// TIA Portal V17 export
// export: Created 2024-09-02T12:50:23.7174179Z, ExportSetting WithDefaults, DisplayName Totally Integrated Automation Portal, DisplayVersion V17, DisplayName TIA Portal Openness, DisplayVersion V17, DisplayName TIA Portal Version Control Interface, DisplayVersion V17, DisplayName STEP 7 Professional, DisplayVersion V17, DisplayName STEP 7 Safety, DisplayVersion V17, DisplayName WinCC Professional, DisplayVersion V17
FUNCTION "AnwFC_StatusStation_OP70" : Void   // FC43, LAD
{ S7_Optimized_Access := 'TRUE' }
VERSION : 0.1
// stored: AutoNumber true, IsIECCheckEnabled false, SetENOAutomatically false, UDAEnableTagReadback false
   VAR_TEMP   // added for the SCL form of the ladder/FBD networks
      _w1 : Bool;
   END_VAR
BEGIN

REGION Network 1: Station Status signals
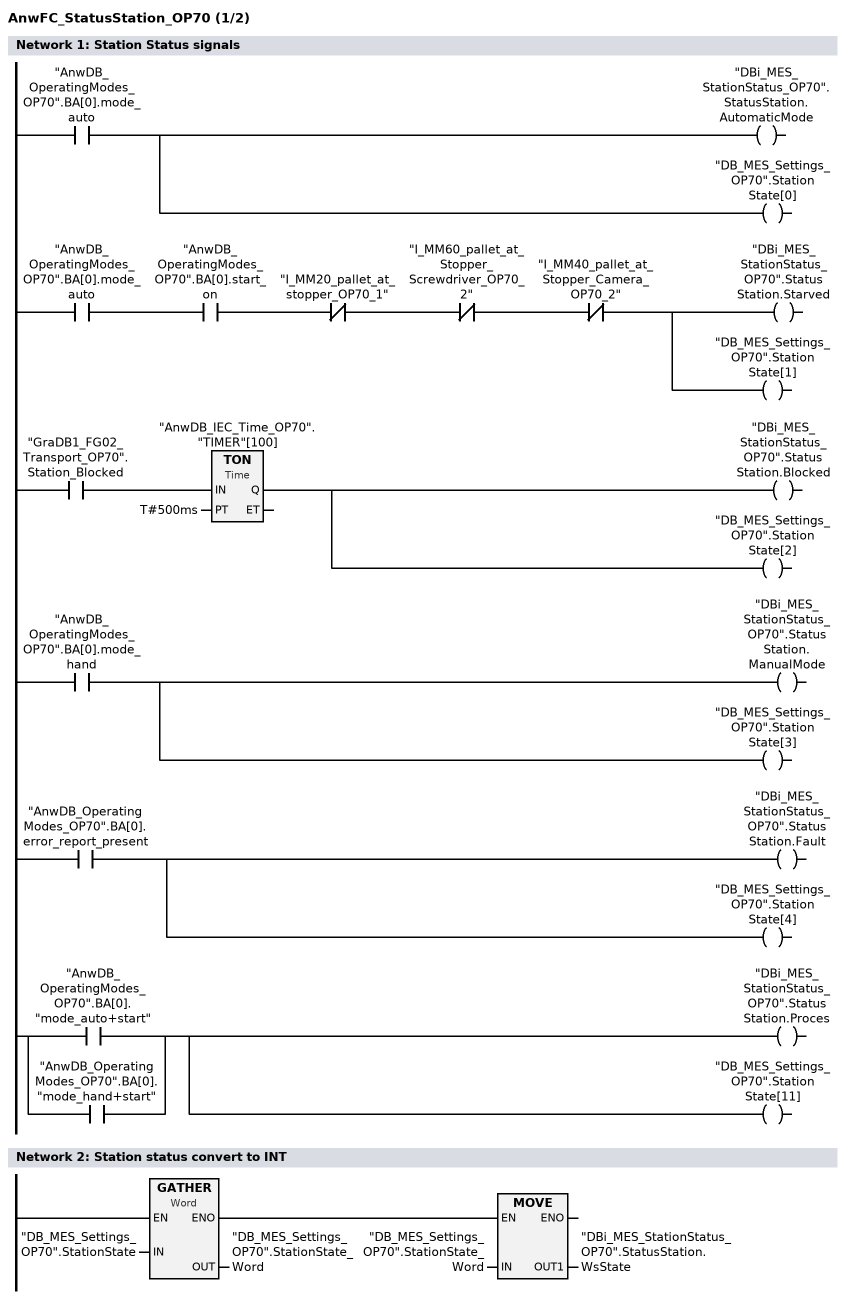
   RUNG wire#powerrail
      Contact( "AnwDB_OperatingModes_OP70".BA[0].mode_auto )
      wire#w1
      Coil( "DBi_MES_StationStatus_OP70".StatusStation.AutomaticMode )
   END_RUNG
   RUNG wire#w1
      Coil( "DB_MES_Settings_OP70".StationState[0] )
   END_RUNG
   RUNG wire#powerrail
      Contact( "AnwDB_OperatingModes_OP70".BA[0].mode_auto )
      Contact( "AnwDB_OperatingModes_OP70".BA[0].start_on )
      I_Contact( "I_MM20_pallet_at_stopper_OP70_1" )
      I_Contact( "I_MM60_pallet_at_Stopper_Screwdriver_OP70_2" )
      I_Contact( "I_MM40_pallet_at_Stopper_Camera_OP70_2" )
      wire#w2
      Coil( "DBi_MES_StationStatus_OP70".StatusStation.Starved )
   END_RUNG
   RUNG wire#w2
      Coil( "DB_MES_Settings_OP70".StationState[1] )
   END_RUNG
   RUNG wire#powerrail
      Contact( "GraDB1_FG02_Transport_OP70".Station_Blocked )
      { S7_Templates := "time_type := Time" } "AnwDB_IEC_Time_OP70"."TIMER"[100].TON(pt := T#500ms, et =>)
      wire#w3
      Coil( "DBi_MES_StationStatus_OP70".StatusStation.Blocked )
   END_RUNG
   RUNG wire#w3
      Coil( "DB_MES_Settings_OP70".StationState[2] )
   END_RUNG
   RUNG wire#powerrail
      Contact( "AnwDB_OperatingModes_OP70".BA[0].mode_hand )
      wire#w4
      Coil( "DBi_MES_StationStatus_OP70".StatusStation.ManualMode )
   END_RUNG
   RUNG wire#w4
      Coil( "DB_MES_Settings_OP70".StationState[3] )
   END_RUNG
   RUNG wire#powerrail
      Contact( "AnwDB_OperatingModes_OP70".BA[0].error_report_present )
      wire#w5
      Coil( "DBi_MES_StationStatus_OP70".StatusStation.Fault )
   END_RUNG
   RUNG wire#w5
      Coil( "DB_MES_Settings_OP70".StationState[4] )
   END_RUNG
   RUNG wire#powerrail
      Contact( "AnwDB_OperatingModes_OP70".BA[0]."mode_auto+start" )
      wire#w6
      Coil( "DBi_MES_StationStatus_OP70".StatusStation.Proces )
   END_RUNG
   RUNG wire#powerrail
      Contact( "AnwDB_OperatingModes_OP70".BA[0]."mode_hand+start" )
   END_RUNG wire#w6
   RUNG wire#w6
      Coil( "DB_MES_Settings_OP70".StationState[11] )
   END_RUNG
   // the same network as SCL:
   "DBi_MES_StationStatus_OP70".StatusStation.AutomaticMode := "AnwDB_OperatingModes_OP70".BA[0].mode_auto;
   "DB_MES_Settings_OP70".StationState[0] := "AnwDB_OperatingModes_OP70".BA[0].mode_auto;
   "DBi_MES_StationStatus_OP70".StatusStation.Starved := "AnwDB_OperatingModes_OP70".BA[0].mode_auto AND "AnwDB_OperatingModes_OP70".BA[0].start_on AND NOT "I_MM20_pallet_at_stopper_OP70_1" AND NOT "I_MM60_pallet_at_Stopper_Screwdriver_OP70_2" AND NOT "I_MM40_pallet_at_Stopper_Camera_OP70_2";
   "DB_MES_Settings_OP70".StationState[1] := "DBi_MES_StationStatus_OP70".StatusStation.Starved;
   "AnwDB_IEC_Time_OP70"."TIMER"[100].TON(IN := "GraDB1_FG02_Transport_OP70".Station_Blocked, PT := T#500ms);
   "DBi_MES_StationStatus_OP70".StatusStation.Blocked := "AnwDB_IEC_Time_OP70"."TIMER"[100].Q;
   "DB_MES_Settings_OP70".StationState[2] := "AnwDB_IEC_Time_OP70"."TIMER"[100].Q;
   "DBi_MES_StationStatus_OP70".StatusStation.ManualMode := "AnwDB_OperatingModes_OP70".BA[0].mode_hand;
   "DB_MES_Settings_OP70".StationState[3] := "AnwDB_OperatingModes_OP70".BA[0].mode_hand;
   "DBi_MES_StationStatus_OP70".StatusStation.Fault := "AnwDB_OperatingModes_OP70".BA[0].error_report_present;
   "DB_MES_Settings_OP70".StationState[4] := "AnwDB_OperatingModes_OP70".BA[0].error_report_present;
   "DBi_MES_StationStatus_OP70".StatusStation.Proces := "AnwDB_OperatingModes_OP70".BA[0]."mode_auto+start" OR "AnwDB_OperatingModes_OP70".BA[0]."mode_hand+start";
   "DB_MES_Settings_OP70".StationState[11] := "DBi_MES_StationStatus_OP70".StatusStation.Proces;
END_REGION

REGION Network 2: Station status convert to INT
   RUNG wire#powerrail
      { S7_Templates := "[dest_type := Word, src_type := Bool]" } GATHER(IN := "DB_MES_Settings_OP70".StationState, OUT => "DB_MES_Settings_OP70".StationState_Word)
      Move(in := "DB_MES_Settings_OP70".StationState_Word, out1 => "DBi_MES_StationStatus_OP70".StatusStation.WsState)
   END_RUNG
   // the same network as SCL:
   GATHER(IN := "DB_MES_Settings_OP70".StationState,
          OUT => "DB_MES_Settings_OP70".StationState_Word,
          ENO => #_w1);
   IF #_w1 THEN
       "DBi_MES_StationStatus_OP70".StatusStation.WsState := "DB_MES_Settings_OP70".StationState_Word;
   END_IF;
END_REGION

REGION Network 3: User EKS_LVL
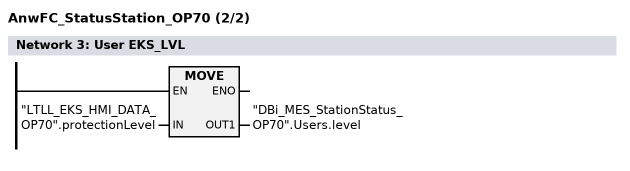
   RUNG wire#powerrail
      Move(in := "LTLL_EKS_HMI_DATA_OP70".protectionLevel, out1 => "DBi_MES_StationStatus_OP70".Users.level)
   END_RUNG
   // the same network as SCL:
   "DBi_MES_StationStatus_OP70".Users.level := "LTLL_EKS_HMI_DATA_OP70".protectionLevel;
END_REGION

REGION Network 4: Error Code
END_REGION
END_FUNCTION
